{attribute addProperty BoxType "EP9521-0020-0000"}
{attribute addProperty Id "A_0025_EP9576_1032_0016EP9576_EEF1625221827.25"}
{attribute addProperty CRC "742428458"}
{attribute addProperty SizeInBites "218"}
{attribute addProperty SizeInBytes "27.25"}
TYPE A_0024_EP9521_0020_0000_2C408F2A EXTENDS EP9521_179A0949 :
STRUCT
	{attribute addProperty Name "A_0025_EP9576_1032_0016"}
	A_0025_EP9576_1032_0016 : EP9576_EEF16252;
END_STRUCT
END_TYPE

(* stored: Version 1.2.0.0, ProductVersion 3.1.4024.9
   DUT A_0024_EP9521_0020_0000_2C408F2A: Id {ccb7f189-6919-41f9-9b60-59382b7ec588} *)
